(* Logix 5000 project; controller Balls vendor 1 type 14 code 149 rev 34.11; software revision 34.00 *)

TASK MainTask (continuous, watchdog 500 ms) : MainProgram

MODULES
   Local : vendor 1 type 14 code 149 (Compact 0, rev 34.11)
      Discrete_IO : Embedded (Compact 1, rev 3.1, Output RPI 20 ms)
END_MODULES

PROGRAM MainProgram   (* main routine MainRoutine *)
VAR
   Ball_in_gravity_chute : ALIAS FOR Local:1:I.Data.5;
   Capacitive_sensor : ALIAS FOR Local:1:I.Data.2;
   ejectpiston1 : ALIAS FOR Local:1:I.Data.0;
   ejectpiston2 : ALIAS FOR Local:1:I.Data.1;
   ejectvalve : ALIAS FOR Local:1:O.Data.0;
   Gate1 : ALIAS FOR Local:1:O.Data.1;
   Gate2 : ALIAS FOR Local:1:O.Data.2;
   inductive_sensor : ALIAS FOR Local:1:I.Data.4;
   Optical_sensor : ALIAS FOR Local:1:I.Data.3;
   Power : BOOL := 1;
   Start : ALIAS FOR Local:1:I.Data.6;
   Stop : ALIAS FOR Local:1:I.Data.7;
   Timer : TIMER := (PRE := 10000);
END_VAR

ROUTINE MainRoutine   (* ladder *)
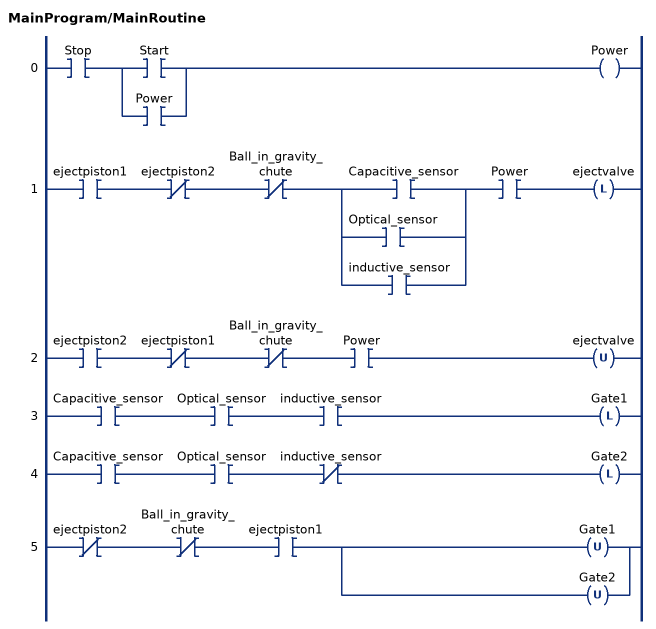
   0: XIC(Stop)[XIC(Start) ,XIC(Power) ]OTE(Power);
   1: XIC(ejectpiston1)XIO(ejectpiston2)XIO(Ball_in_gravity_chute)[XIC(Capacitive_sensor) ,XIC(Optical_sensor) ,XIC(inductive_sensor) ]XIC(Power)OTL(ejectvalve);
   2: XIC(ejectpiston2)XIO(ejectpiston1)XIO(Ball_in_gravity_chute)XIC(Power)OTU(ejectvalve);
   3: XIC(Capacitive_sensor)XIC(Optical_sensor)XIC(inductive_sensor)OTL(Gate1);
   4: XIC(Capacitive_sensor)XIC(Optical_sensor)XIO(inductive_sensor)OTL(Gate2);
   5: XIO(ejectpiston2)XIO(Ball_in_gravity_chute)XIC(ejectpiston1)[OTU(Gate1) ,OTU(Gate2) ];
END_ROUTINE
END_PROGRAM
